FUNCTION_BLOCK FB_StewartInterface
VAR_INPUT
	// Stewart Operation 
	bStop : BOOL;
	bReset : BOOL;
	bResetScale : BOOL;
	bStart : BOOL;
	eModeCmd : E_StewartMode;
	
	// Remote data input
	bRemoteActive : BOOL := FALSE;
	uRemote : ARRAY [0..5] OF LREAL;
	
END_VAR
VAR_OUTPUT
	bError : BOOL;
	bBusy : BOOL := FALSE;
	bReady : BOOL := FALSE;
	eState : E_StewartState;
	eStatus : E_StewartStatus;
	eOpMode : E_StewartOpMode;
	eMode : E_StewartMode;
	
	// Feedback data
	feedback : ST_FeedbackStewart;
	
	(*
	eta : ARRAY [0..5] OF LREAL;
	eta_t : ARRAY [0..5] OF LREAL;
	eta_tt : ARRAY [0..5] OF LREAL;
	*)
	
END_VAR
VAR	
	// Hydro Simualator
	hydro : FB_HydroSimulator(0);
	
	// Stewart positon input
	u : ARRAY [0..5] OF LREAL;
	u_t : ARRAY [0..5] OF LREAL;
	uOld : ARRAY [0..5] OF LREAL;
	
	// Stewart soft motion
	fbSoftMotion : ARRAY [0..5] OF FB_SoftMotion;
	
	// Limted stewart setpoints
	etaRef : ARRAY [0..5] OF LREAL;
	etaRef_t : ARRAY [0..5] OF LREAL;
	etaRef_tt : ARRAY [0..5] OF LREAL;
	etaRefOld : ARRAY [0..5] OF LREAL;

	// Sine wave data
	etaSine : ARRAY [0..5] OF LREAL;
	etaSine_t : ARRAY [0..5] OF LREAL;
	etaSine_tt : ARRAY [0..5] OF LREAL;
	
	// Udp connection
	udpClient : FB_UdpClientRT('', 0, 0, 0, 0, 0, 0);	// Dummy constructor

	{attribute 'tc_no_symbol'}
	eCmnd : E_StewartCommand;
	{attribute 'tc_no_symbol'}
	rxUdp : ST_RxUdpStewart;
	{attribute 'tc_no_symbol'}
	txUdp : ST_TxUdpStewart;
	
	// Hmi connection
	txHmi : ST_TxHmiStewart;
	
	// Udp activity monitoring
	bActive : BOOL;
	frame : UDINT := 0;
	frameOld : UDINT := 0;
	frameLoss : UDINT := 0;
	
	// Task monitoring
	fbGetCurrentTaskIdx : GETCURTASKINDEX;
	bCycleTimeExceeded : BOOL;
	nCycleCount : UDINT;
	Ts : LREAL;
	t : LREAL := 0.0;
	
	// Sine Generator Settings
	sineAmplitude : ARRAY [0..5] OF LREAL := [0, 0, 0.2, 2.0/180.0*PI, 2.0/180.0*PI, 0];
	sineOmega : ARRAY [0..5] OF LREAL := [0.6283, 0.6283, 0.6283, 0.6283, 0.6283, 0.6283];
	sinePhase : ARRAY [0..5] OF LREAL;

	// Zero eta
	{attribute 'tc_no_symbol'}
	etaZeros : ARRAY [0..5] OF LREAL;
	
	// Max/min settings
	etaRefMin : ARRAY [0..5] OF LREAL;
	etaRefMax : ARRAY [0..5] OF LREAL;
END_VAR

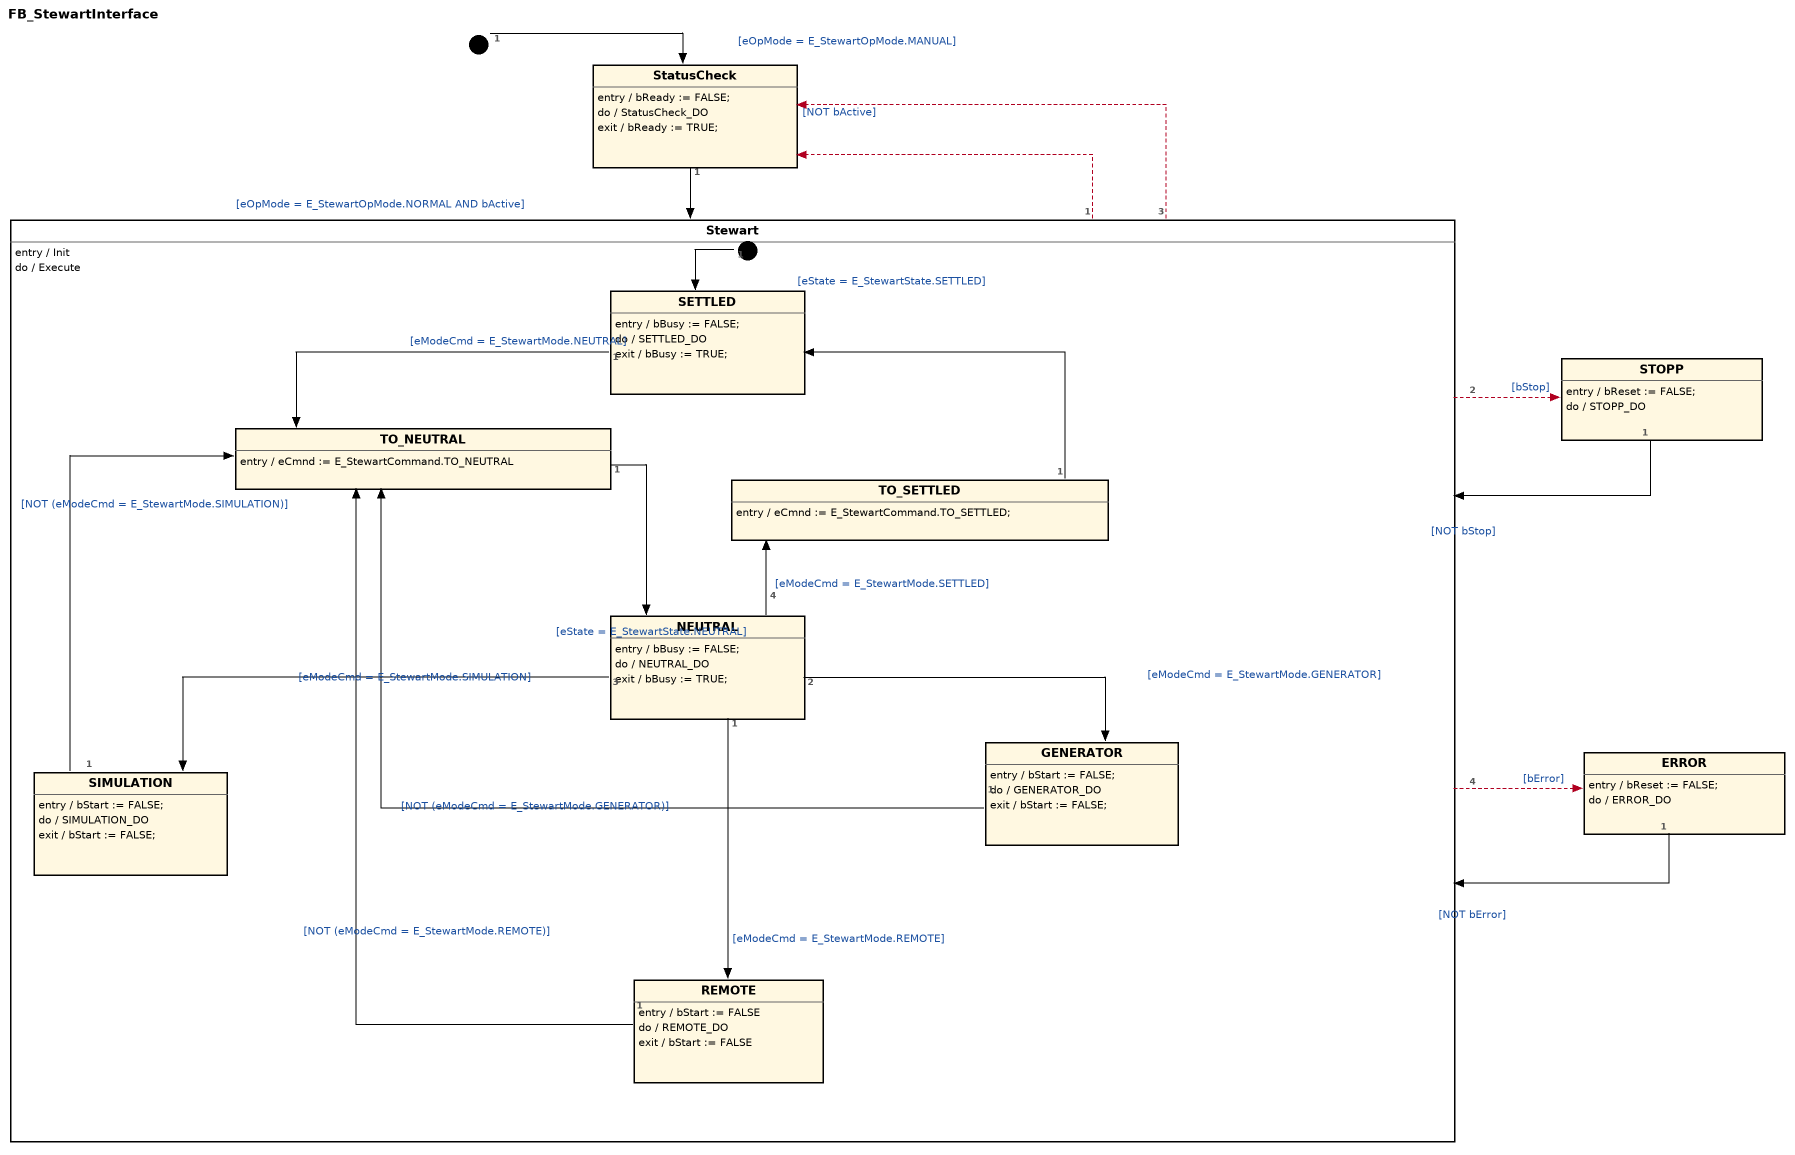
STATECHART ST_StewartInterface  // abortable
    START StartState1
    STATE StatusCheck
        entry / bReady := FALSE;
        do / StatusCheck_DO
        exit / bReady := TRUE;
    COMPOSITE STATE Stewart
        entry / Init
        do / Execute
        START StartState2
        STATE SETTLED
            entry / bBusy := FALSE;
            do / SETTLED_DO
            exit / bBusy := TRUE;
        STATE TO_NEUTRAL
            entry / eCmnd := E_StewartCommand.TO_NEUTRAL
        STATE TO_SETTLED
            entry / eCmnd := E_StewartCommand.TO_SETTLED;
        STATE NEUTRAL
            entry / bBusy := FALSE;
            do / NEUTRAL_DO
            exit / bBusy := TRUE;
        STATE GENERATOR
            entry / bStart := FALSE;
            do / GENERATOR_DO
            exit / bStart := FALSE;
        STATE SIMULATION
            entry / bStart := FALSE;
            do / SIMULATION_DO
            exit / bStart := FALSE;
        STATE REMOTE
            entry / bStart := FALSE
            do / REMOTE_DO
            exit / bStart := FALSE
        StartState2 -> SETTLED  // priority 1, on completion
        SETTLED -> TO_NEUTRAL [eModeCmd = E_StewartMode.NEUTRAL] // priority 1
        TO_NEUTRAL -> NEUTRAL [eState = E_StewartState.NEUTRAL] // priority 1
        TO_SETTLED -> SETTLED [eState = E_StewartState.SETTLED] // priority 1
        NEUTRAL -> REMOTE [eModeCmd = E_StewartMode.REMOTE] // priority 1
        NEUTRAL -> GENERATOR [eModeCmd = E_StewartMode.GENERATOR] // priority 2
        NEUTRAL -> SIMULATION [eModeCmd = E_StewartMode.SIMULATION] // priority 3
        NEUTRAL -> TO_SETTLED [eModeCmd = E_StewartMode.SETTLED] // priority 4
        GENERATOR -> TO_NEUTRAL [NOT (eModeCmd = E_StewartMode.GENERATOR)] // priority 1
        SIMULATION -> TO_NEUTRAL [NOT (eModeCmd = E_StewartMode.SIMULATION)] // priority 1
        REMOTE -> TO_NEUTRAL [NOT (eModeCmd = E_StewartMode.REMOTE)] // priority 1
    END_STATE
    STATE STOPP
        entry / bReset := FALSE;
        do / STOPP_DO
    STATE ERROR
        entry / bReset := FALSE;
        do / ERROR_DO
    StartState1 -> StatusCheck  // priority 1, on completion
    StatusCheck -> Stewart [eOpMode = E_StewartOpMode.NORMAL AND bActive] // priority 1
    Stewart -> StatusCheck [NOT bActive] // priority 1, exception
    Stewart -> STOPP [bStop] // priority 2, exception
    Stewart -> StatusCheck [eOpMode = E_StewartOpMode.MANUAL] // priority 3, exception
    Stewart -> ERROR [bError] // priority 4, exception
    STOPP -> Stewart [NOT bStop] // priority 1
    ERROR -> Stewart [NOT bError] // priority 1
END_STATECHART

METHOD decode_E_StewartOpMode : E_StewartOpMode
VAR_INPUT
	motionStatus : UDINT;
END_VAR
VAR
	mask : UDINT;
	n : USINT;
END_VAR

mask := 16#FF000000 AND motionStatus;
n := UDINT_TO_USINT(SHR(mask, 6));

(*
CASE mask OF
	16#00000000 :
		eResult := E_StewartOpMode.MANUAL;
		
	16#01000000 :
		eResult := E_StewartOpMode.NORMAL;
	
END_CASE
*)
END_METHOD

METHOD PRIVATE decode_E_StewartState : E_StewartState
VAR_INPUT
	motionStatus : UDINT;
END_VAR
VAR
	mask : UDINT;
	eResult : E_StewartState;
END_VAR
// PDF: Motion System Ethernet Interface p.18

mask := 16#0000000F AND motionStatus;

CASE mask OF
	16#00000000 : 
		eResult := E_StewartState.TRANSIT;
		
	16#00000001 : 
		eResult := E_StewartState.OFF;
		
	16#00000002 : 
		eResult := E_StewartState.SETTLED;
		
	16#00000003 : 
		eResult := E_StewartState.OIL_HEATING;
		
	16#00000004 : 
		eResult := E_StewartState.NEUTRAL;
		
	16#00000005 : 
		eResult := E_StewartState.NEUTRAL_FREEZE;
		
	16#00000008 : 
		eResult := E_StewartState.ENGAGED;
		
	16#00000009 : 
		eResult := E_StewartState.ENGAGED_FREEZE;
	
END_CASE

decode_E_StewartState := eResult;
END_METHOD

METHOD decode_E_StewartStatus : E_StewartStatus
VAR_INPUT
	motionStatus : UDINT;
END_VAR
VAR
	mask : UDINT;
	eResult : E_StewartStatus;
END_VAR

mask := 16#000000F0 AND motionStatus;

CASE mask OF
	16#00000000 :
		eResult := E_StewartStatus.SYSTEM_OK;
		
	16#01000040 :
		eResult := E_StewartStatus.WARNING;
		
	16#01000080 :
		eResult := E_StewartStatus.ERROR;
	
END_CASE

decode_E_StewartStatus := eResult;
END_METHOD

METHOD PRIVATE ERROR_DO : BOOL
VAR_INPUT
END_VAR
// Wait for SYSTEM_OK and return to settled
IF eStatus = E_StewartStatus.SYSTEM_OK THEN
	eModeCmd := E_StewartMode.SETTLED;
	eCmnd := E_StewartCommand.TO_SETTLED;

	bError := FALSE;
	
END_IF

// Check for bReset request and acknowledge fault
IF bReset THEN
	eCmnd := E_StewartCommand.ACK_FAULT;
	bReset := FALSE;
END_IF

// Execute main thread
Execute();
END_METHOD

METHOD PRIVATE Execute : BOOL
VAR_INPUT
END_VAR
VAR

	i: INT;
	
	nState : DWORD;
	nStatus : DWORD;
	nOpMode : DWORD;
	
	amp : LREAL;
	omega : LREAL;
	phi : LREAL;
	
	(*
	// Velocity boundary
	qMin : ARRAY [0..5] OF LREAL := [-0.2, -0.2, -0.2, -5.0/180.0*PI, -5.0/180.0*PI, -5.0/180.0*PI];
	qMax : ARRAY [0..5] OF LREAL := [ 0.2,  0.2,  0.2,  5.0/180.0*PI,  5.0/180.0*PI,  5.0/180.0*PI];
	V : ARRAY [0..5] OF LREAL := [6(1.0)];
	A : ARRAY [0..5] OF LREAL := [6(1.0)];
	stVelocityBoundary : ARRAY [0..5] OF ST_VelocityBoundary;
	*)
	
	
	
END_VAR
// Task monitoring
fbGetCurrentTaskIdx();
bCycleTimeExceeded := _TaskInfo[fbGetCurrentTaskIdx.index].CycleTimeExceeded;
nCycleCount := _TaskInfo[fbGetCurrentTaskIdx.index].CycleCount;
Ts := UDINT_TO_LREAL(_TaskInfo[fbGetCurrentTaskIdx.index].CycleTime/10)/1E6;

// Hydro Simualtor Scale reset logic
IF bResetScale THEN
	CASE eMode OF
		E_StewartMode.SETTLED, E_StewartMode.NEUTRAL :
			hydro.stInput.bReset := TRUE;
			bResetScale := FALSE;

		ELSE
			eModeCmd := E_StewartMode.NEUTRAL;				
	
	END_CASE
END_IF

// Hydro simulator
IF hydro.State = TCOM_STATE.TCOM_STATE_OP THEN
	hydro.Execute();
	hydro.stInput.bReset := FALSE;
	
END_IF

// Increment Timer
t := t + Ts;

// Set control command
txUdp.CMND := eCmnd;


(* // SOFT INPUT
// Set soft motion input
IF Ts > 0 THEN
	FOR i := 0 TO 5 DO
		// Get speed by numerical differentiation
		u_t[i] := (u[i] - uOld[i])/Ts;
		uOld[i] := u[i];
		
		fbSoftMotion[i](
			Ts := Ts,
			qRef_t := u_t[i]
		);
		
		etaRef[i] := fbSoftMotion[i].q;
		etaRef_t[i] := fbSoftMotion[i].q_t;
		
		
		
		(*
		// Apply velocity boundary
		stVelocityBoundary[i] := F_VelocityBoundary(etaRef[i], qMin[i], qMax[i], V[i], A[i], Ts);
		
		// Limit Velocity
		
		etaRef_t[i] := MAX(etaRef_t[i], stVelocityBoundary[i].qMin_t);
		etaRef_t[i] := MIN(etaRef_t[i], stVelocityBoundary[i].qMax_t);

		// Apply numerical integration based on etaRef_t
		etaRef[i] := etaRef[i] + etaRef_t[i]*Ts;

		// Absolute postion constraint
		etaRef[i] := MAX(etaRef[i], qMin[i]);
		etaRef[i] := MIN(etaRef[i], qMax[i]);
		
		// TODO: Numerical acceleration?
		*)
		
	END_FOR
	
END_IF
*)

// NO SOF STOP Motion
FOR i := 0 TO 5 DO
	etaRef[i] := LIMIT(etaRefMin[i], u[i], etaRefMax[i]);
	etaRef_t[i] := 0.0;
 
END_FOR

// Assign motion to Stewart
txUdp.X_EXTRA 			:= LREAL_TO_REAL(etaRef[0]);
txUdp.Y_EXTRA 			:= LREAL_TO_REAL(etaRef[1]);
txUdp.Z_EXTRA 			:= LREAL_TO_REAL(etaRef[2]);
txUdp.PHI_EXTRA 		:= LREAL_TO_REAL(etaRef[3]);
txUdp.THETA_EXTRA 		:= LREAL_TO_REAL(etaRef[4]);
txUdp.PSI_EXTRA 		:= LREAL_TO_REAL(etaRef[5]);

txUdp.X_EXTRA_DOT		:= LREAL_TO_REAL(etaRef_t[0]);
txUdp.Y_EXTRA_DOT		:= LREAL_TO_REAL(etaRef_t[1]);
txUdp.Z_EXTRA_DOT		:= LREAL_TO_REAL(etaRef_t[2]);
txUdp.PHI_EXTRA_DOT		:= LREAL_TO_REAL(etaRef_t[3]);
txUdp.THETA_EXTRA_DOT	:= LREAL_TO_REAL(etaRef_t[4]);
txUdp.PSI_EXTRA_DOT		:= LREAL_TO_REAL(etaRef_t[5]);

txUdp.X_EXTRA_DDOT		:= 0.0;
txUdp.Y_EXTRA_DDOT		:= 0.0;
txUdp.Z_EXTRA_DDOT		:= 0.0;
txUdp.PHI_EXTRA_DDOT	:= 0.0;
txUdp.THETA_EXTRA_DDOT	:= 0.0;
txUdp.PSI_EXTRA_DDOT	:= 0.0;


// Update udpClient
udpClient();

// Unamsk Motion_Status signal
nState	:= 16#0000000F AND rxUdp.Motion_Status;
nStatus	:= 16#000000F0 AND rxUdp.Motion_Status;
nOpMode := 16#FF000000 AND rxUdp.Motion_Status;

// Shift for USINT conversion
nState 	:= SHR(nState, 0*4);
nStatus := SHR(nStatus, 1*4);
nOpMode := SHR(nOpMode, 6*4);

// Enum(USINT) typecast
MEMCPY(ADR(eState), ADR(nState), SIZEOF(eState));
MEMCPY(ADR(eStatus), ADR(nStatus), SIZEOF(eStatus));
MEMCPY(ADR(eOpMode), ADR(nOpMode), SIZEOF(eOpMode));

// Error/Warning check
IF (eStatus <> E_StewartStatus.SYSTEM_OK) THEN
	bError := TRUE;;
END_IF

// Check activity
frame := rxUdp.Frame_Count;
IF frame <> frameOld THEN
	// Update frame old
	frameOld := frame;
	
	// Reset frameLoss
	frameLoss := 0;
ELSE
	// Count frame losses
	frameLoss := frameLoss + 1;
END_IF

// Set activity status after 1 second given 5ms in ms
IF frameLoss > 200 THEN
	bActive := FALSE;
ELSE
	bActive := TRUE;
END_IF

// Feedback data
feedback.eta[0] := REAL_TO_LREAL(rxUdp.Actual_platform_position_surge);
feedback.eta[1] := REAL_TO_LREAL(rxUdp.Actual_platform_position_sway);
feedback.eta[2] := REAL_TO_LREAL(rxUdp.Actual_platform_position_heave);
feedback.eta[3] := REAL_TO_LREAL(rxUdp.Actual_platform_position_roll);
feedback.eta[4] := REAL_TO_LREAL(rxUdp.Actual_platform_position_pitch);
feedback.eta[5] := REAL_TO_LREAL(rxUdp.Actual_platform_position_yaw);

feedback.eta_t[0] := REAL_TO_LREAL(rxUdp.Actual_platform_velocity_surge);
feedback.eta_t[1] := REAL_TO_LREAL(rxUdp.Actual_platform_velocity_sway);
feedback.eta_t[2] := REAL_TO_LREAL(rxUdp.Actual_platform_velocity_heave);
feedback.eta_t[3] := REAL_TO_LREAL(rxUdp.Actual_platform_velocity_roll);
feedback.eta_t[4] := REAL_TO_LREAL(rxUdp.Actual_platform_velocity_pitch);
feedback.eta_t[5] := REAL_TO_LREAL(rxUdp.Actual_platform_velocity_yaw);

feedback.eta_tt[0] := REAL_TO_LREAL(rxUdp.Actual_platform_acceleration_surge);
feedback.eta_tt[1] := REAL_TO_LREAL(rxUdp.Actual_platform_acceleration_sway);
feedback.eta_tt[2] := REAL_TO_LREAL(rxUdp.Actual_platform_acceleration_heave);
feedback.eta_tt[3] := REAL_TO_LREAL(rxUdp.Actual_platform_acceleration_roll);
feedback.eta_tt[4] := REAL_TO_LREAL(rxUdp.Actual_platform_acceleration_pitch);
feedback.eta_tt[5] := REAL_TO_LREAL(rxUdp.Actual_platform_acceleration_yaw);

// Update global Hmi data
IF bActive THEN
	txHmi.status := 1;
ELSE
	txHmi.status := 0;
END_IF

txHmi.eta[0] := rxUdp.Actual_platform_position_surge;
txHmi.eta[1] := rxUdp.Actual_platform_position_sway;
txHmi.eta[2] := rxUdp.Actual_platform_position_heave;
txHmi.eta[3] := rxUdp.Actual_platform_position_roll;
txHmi.eta[4] := rxUdp.Actual_platform_position_pitch;
txHmi.eta[5] := rxUdp.Actual_platform_position_yaw;

txHmi.etaRef[0] := rxUdp.Platform_setpoint_surge;
txHmi.etaRef[1] := rxUdp.Platform_setpoint_sway;
txHmi.etaRef[2] := rxUdp.Platform_setpoint_heave;
txHmi.etaRef[3] := rxUdp.Platform_setpoint_roll;
txHmi.etaRef[4] := rxUdp.Platform_setpoint_pitch;
txHmi.etaRef[5] := rxUdp.Platform_setpoint_yaw;

txHmi.cyl[0] := rxUdp.Actual_position_actuator_1;
txHmi.cyl[1] := rxUdp.Actual_position_actuator_2;
txHmi.cyl[2] := rxUdp.Actual_position_actuator_3;
txHmi.cyl[3] := rxUdp.Actual_position_actuator_4;
txHmi.cyl[4] := rxUdp.Actual_position_actuator_5;
txHmi.cyl[5] := rxUdp.Actual_position_actuator_6;

FOR i := 0 TO 5 DO
	txHmi.dofScale[i] := LREAL_TO_REAL(hydro.stOutput.scale[i]);
END_FOR
END_METHOD

METHOD FB_exit : BOOL
VAR_INPUT
	bInCopyCode : BOOL; // if TRUE, the exit method is called for exiting an instance that is copied afterwards (online change).
END_VAR
END_METHOD

METHOD FB_init : BOOL
VAR_INPUT
	bInitRetains : BOOL; // if TRUE, the retain variables are initialized (warm start / cold start)
	bInCopyCode : BOOL;  // if TRUE, the instance afterwards gets moved into the copy code (online change)
	
	// Init variables
	_remoteIpAddr : T_Ipv4Addr;
	_remotePort : UINT;
	_localPort : UINT;
	oid : OTCID;
	

END_VAR
// Initilize udpClient
udpClient.FB_init(
	bInitRetains,
	bInCopyCode,
	_remoteIpAddr,
	_remotePort,
	_localPort,
	SIZEOF(rxUdp),
	ADR(rxUdp),
	SIZEOF(txUdp),
	ADR(txUdp)
);

// TcCOM adress
hydro.FB_init(bInitRetains, bInCopyCode, oid);

// EM8000
IF _remotePort = 50030 THEN
	rxUdp.Actual_platform_position_heave := 0.9986208;
	
	// Max/min strokes
	etaRefMin[0] := -0.2;
	etaRefMin[1] := -0.2;
	etaRefMin[2] := -0.6;
	etaRefMin[3] := -5.0/180*PI;
	etaRefMin[4] := -5.0/180*PI;
	etaRefMin[5] := -10.0/180*PI;
	
	etaRefMax[0] := 0.2;
	etaRefMax[1] := 0.2;
	etaRefMax[2] := 0.6;
	etaRefMax[3] := 5.0/180*PI;
	etaRefMax[4] := 5.0/180*PI;
	etaRefMax[5] := 10.0/180*PI;
END_IF

// EM15000
IF _remotePort = 50031 THEN
	rxUdp.Actual_platform_position_heave := 0.4663845;
	
	// Max/min strokes
	etaRefMin[0] := -0.15;
	etaRefMin[1] := -0.15;
	etaRefMin[2] := -0.3;
	etaRefMin[3] := -5.0/180*PI;
	etaRefMin[4] := -5.0/180*PI;
	etaRefMin[5] := -5.0/180*PI;
	
	etaRefMax[0] := 0.15;
	etaRefMax[1] := 0.15;
	etaRefMax[2] := 0.3;
	etaRefMax[3] := 5.0/180*PI;
	etaRefMax[4] := 5.0/180*PI;
	etaRefMax[5] := 5.0/180*PI;
END_IF
END_METHOD

METHOD FB_reinit : BOOL
VAR_INPUT
END_VAR
END_METHOD

METHOD PRIVATE GENERATOR_DO : BOOL
VAR_INPUT
END_VAR
VAR
	i : UINT;
	
	amp : LREAL;
	omega : LREAL;
	phi : LREAL;
	
END_VAR

// Apply sine generator input
FOR i := 0 TO 5 DO
	// Sine signals
	amp := sineAmplitude[i];
	omega := sineOmega[i];
	phi := sinePhase[i];
	
	u[i] := amp*SIN(omega*t + phi);
	
END_FOR


IF bStart THEN
	eCmnd := E_StewartCommand.TO_ENGAGED;
	
ELSE
	eCmnd := E_StewartCommand.TO_NEUTRAL;
	
END_IF

// Set mode
eMode := E_StewartMode.GENERATOR;
END_METHOD

METHOD PRIVATE Init
VAR_INPUT
END_VAR
// Do init here
END_METHOD

METHOD PRIVATE NEUTRAL_DO : BOOL
VAR_INPUT
END_VAR
VAR
	i : UINT;
END_VAR
// Zero input
etaRef := etaZeros;
etaRef_t := etaZeros;
etaRef_tt := etaZeros;

// Set mode
eMode := E_StewartMode.NEUTRAL;
END_METHOD

METHOD PRIVATE REMOTE_DO : BOOL
VAR_INPUT
END_VAR
VAR
	i : UINT;
	bLimitExceeded : BOOL;
END_VAR
// Check input
FOR i := 0 TO 5 DO
	IF (u[i] < etaRefMin[i]) OR (u[i] > etaRefMax[i]) THEN
		bLimitExceeded := TRUE;
		
	END_IF
END_FOR

// Set input from remote
u := uRemote;

// Enagage and disengage if remote is active
IF bStart AND bRemoteActive AND NOT bLimitExceeded THEN
	eCmnd := E_StewartCommand.TO_ENGAGED;
	
ELSE
	eCmnd := E_StewartCommand.TO_NEUTRAL;
	
END_IF


// Set mode
eMode := E_StewartMode.REMOTE;
END_METHOD

METHOD PRIVATE SETTLED_DO : BOOL
VAR_INPUT
END_VAR
VAR
	i : UINT;
END_VAR
// Zero input
etaRef := etaZeros;
etaRef_t := etaZeros;
etaRef_tt := etaZeros;


eMode := E_StewartMode.SETTLED;
END_METHOD

METHOD PRIVATE SIMULATION_DO : BOOL
VAR_INPUT
END_VAR
// Apply simulator output
u := hydro.stOutput.eta;

IF bStart THEN
	eCmnd := E_StewartCommand.TO_ENGAGED;
	
ELSE
	eCmnd := E_StewartCommand.TO_NEUTRAL;
	
END_IF
			

// Set mode
eMode := E_StewartMode.SIMULATION;
END_METHOD

METHOD PRIVATE StatusCheck_DO : BOOL
VAR_INPUT
END_VAR
eModeCmd := E_StewartMode.SETTLED;
eCmnd := E_StewartCommand.TO_SETTLED;

Execute();
END_METHOD

METHOD PRIVATE Stewart_DO : BOOL
VAR_INPUT
END_VAR

VAR
	i: INT;
END_VAR



// Execute Main thread 
Execute();
END_METHOD

METHOD PRIVATE STOPP_DO : BOOL
VAR_INPUT
END_VAR
// Got to settled in case of stop
eModeCmd := E_StewartMode.SETTLED;
eCmnd := E_StewartCommand.TO_SETTLED;
	 
// Execute main thread
Execute();

// Reset stop
IF (eStatus = E_StewartStatus.SYSTEM_OK) AND bReset THEN
	bStop := FALSE;
	
END_IF
END_METHOD

END_FUNCTION_BLOCK

(* stored: Version 1.1.0.1, ProductVersion 3.1.4022.18
   POU FB_StewartInterface: Id {bc1132f0-30a6-41f8-8816-fcd499a79e5c}, SpecialFunc None
   Method decode_E_StewartOpMode: Id {aeed7a95-8ef5-47a2-87d9-187ad2fce3da}
   Method decode_E_StewartState: Id {e4d78dc9-868d-41d9-8edb-2d85943c11a0}
   Method decode_E_StewartStatus: Id {bbaee5fb-4eca-4cf3-9659-16a29517b6f5}
   Method ERROR_DO: Id {4a61e0e3-a4c6-4d6d-8f96-df1f66850830}
   Method Execute: Id {7ab70c3b-60b3-4238-ba48-85e0dc447c49}
   Method FB_exit: Id {9bed94a0-b2f9-4c8b-9085-b30806c38f7e}
   Method FB_init: Id {c61434a5-8a62-405e-832e-838499c788e2}
   Method FB_reinit: Id {0d8df33c-9ef8-4c5e-ab3a-f88ad66fdbff}
   Method GENERATOR_DO: Id {56942693-b597-4c5f-bdcd-afda718bb866}
   Method Init: Id {15cd2314-2942-4ebe-a279-270379030e94}
   Method NEUTRAL_DO: Id {69231ff7-e79a-4faa-b660-c71db9a3b5fc}
   Method REMOTE_DO: Id {60908887-7e2a-47de-881c-86e8e5d8344f}
   Method SETTLED_DO: Id {3f622d4b-3977-4a1f-9053-5c946b26f676}
   Method SIMULATION_DO: Id {c4950ba8-bec0-4ee1-aa4a-7e027c541c4f}
   Method StatusCheck_DO: Id {a39a77ba-2cc3-4587-a018-d8ce79cb4e47}
   Method Stewart_DO: Id {3f4bcd7a-1198-44f9-8097-0a0c8b8727c7}
   Method STOPP_DO: Id {c0f5e363-81aa-4e1d-ba41-5ee852d3c92a} *)
